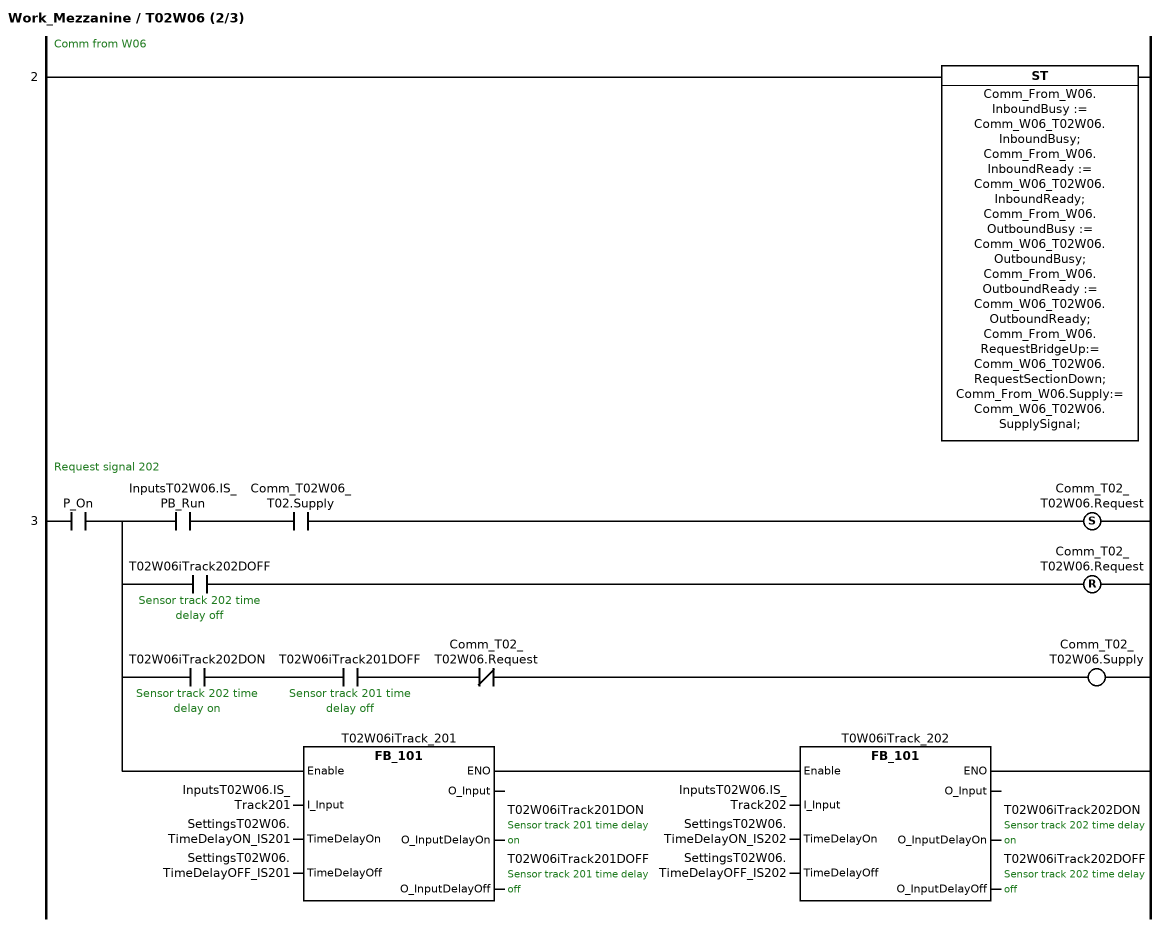
(* [picture p102: Work_Mezzanine / T02W06, rungs 2-3] *)
(* Rung 2: Comm from W06 *)
Comm_From_W06.InboundBusy := Comm_W06_T02W06.InboundBusy;
Comm_From_W06.InboundReady := Comm_W06_T02W06.InboundReady;
Comm_From_W06.OutboundBusy := Comm_W06_T02W06.OutboundBusy;
Comm_From_W06.OutboundReady := Comm_W06_T02W06.OutboundReady;
Comm_From_W06.RequestBridgeUp:= Comm_W06_T02W06.RequestSectionDown;
Comm_From_W06.Supply:= Comm_W06_T02W06.SupplySignal;
(* Rung 3: Request signal 202 *)
IF P_On AND InputsT02W06.IS_PB_Run AND Comm_T02W06_T02.Supply THEN
    Comm_T02_T02W06.Request := TRUE;
END_IF;
IF P_On AND T02W06iTrack202DOFF THEN Comm_T02_T02W06.Request := FALSE; END_IF;
Comm_T02_T02W06.Supply := P_On AND T02W06iTrack202DON AND T02W06iTrack201DOFF AND NOT Comm_T02_T02W06.Request;
T02W06iTrack_201(Enable := P_On, I_Input := InputsT02W06.IS_Track201, TimeDelayOn := SettingsT02W06.TimeDelayON_IS201, TimeDelayOff := SettingsT02W06.TimeDelayOFF_IS201, O_InputDelayOn => T02W06iTrack201DON, O_InputDelayOff => T02W06iTrack201DOFF);
T0W06iTrack_202(Enable := T02W06iTrack_201.ENO, I_Input := InputsT02W06.IS_Track202, TimeDelayOn := SettingsT02W06.TimeDelayON_IS202, TimeDelayOff := SettingsT02W06.TimeDelayOFF_IS202, O_InputDelayOn => T02W06iTrack202DON, O_InputDelayOff => T02W06iTrack202DOFF);

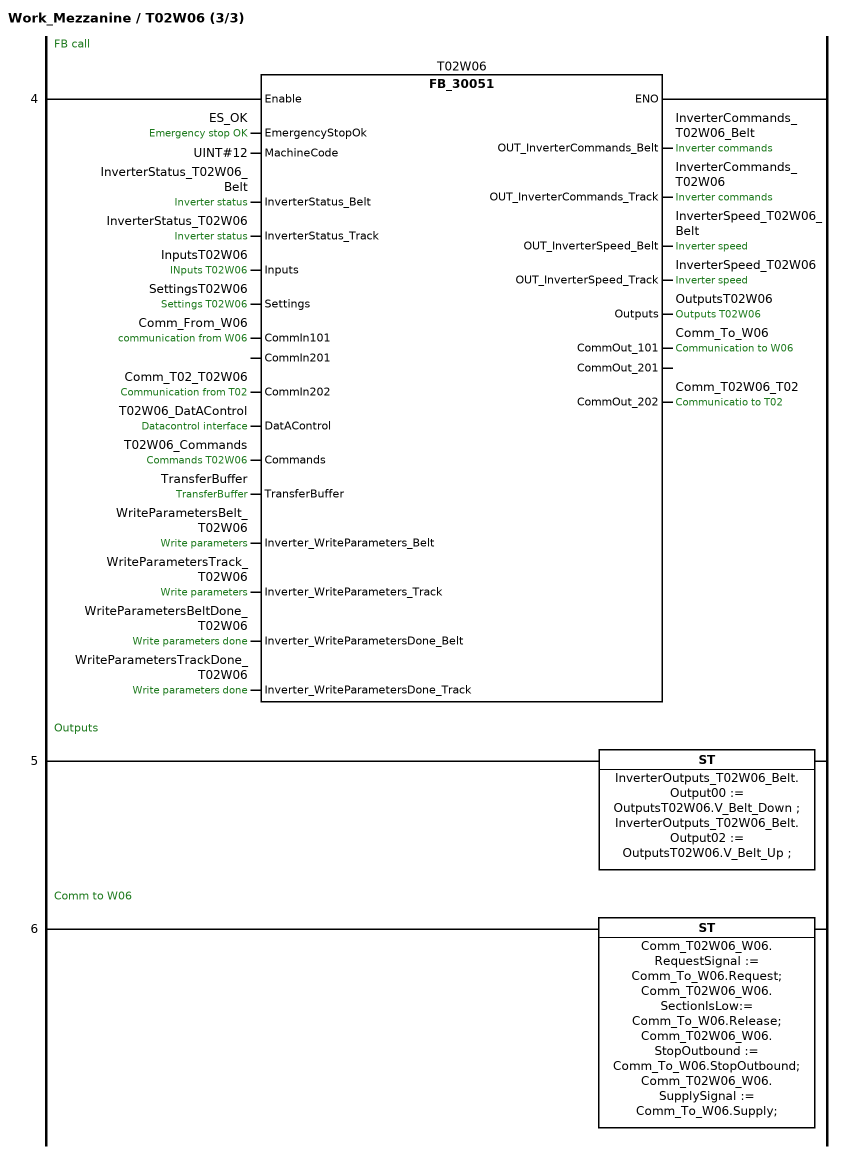
(* Rung 4: FB call *)
T02W06(Enable := TRUE, EmergencyStopOk := ES_OK, MachineCode := UINT#12, InverterStatus_Belt := InverterStatus_T02W06_Belt, InverterStatus_Track := InverterStatus_T02W06, Inputs := InputsT02W06, Settings := SettingsT02W06, CommIn101 := Comm_From_W06, CommIn202 := Comm_T02_T02W06, DatAControl := T02W06_DatAControl, Commands := T02W06_Commands, TransferBuffer := TransferBuffer, Inverter_WriteParameters_Belt := WriteParametersBelt_T02W06, Inverter_WriteParameters_Track := WriteParametersTrack_T02W06, Inverter_WriteParametersDone_Belt := WriteParametersBeltDone_T02W06, Inverter_WriteParametersDone_Track := WriteParametersTrackDone_T02W06, OUT_InverterCommands_Belt => InverterCommands_T02W06_Belt, OUT_InverterCommands_Track => InverterCommands_T02W06, OUT_InverterSpeed_Belt => InverterSpeed_T02W06_Belt, OUT_InverterSpeed_Track => InverterSpeed_T02W06, Outputs => OutputsT02W06, CommOut_101 => Comm_To_W06, CommOut_202 => Comm_T02W06_T02);
(* Rung 5: Outputs *)
InverterOutputs_T02W06_Belt.Output00 := OutputsT02W06.V_Belt_Down ;
InverterOutputs_T02W06_Belt.Output02 := OutputsT02W06.V_Belt_Up ;
(* Rung 6: Comm to W06 *)
Comm_T02W06_W06.RequestSignal := Comm_To_W06.Request;
Comm_T02W06_W06.SectionIsLow:= Comm_To_W06.Release;
Comm_T02W06_W06.StopOutbound := Comm_To_W06.StopOutbound;
Comm_T02W06_W06.SupplySignal := Comm_To_W06.Supply;

(* Section T02W07: ladder, written here as Structured Text *)

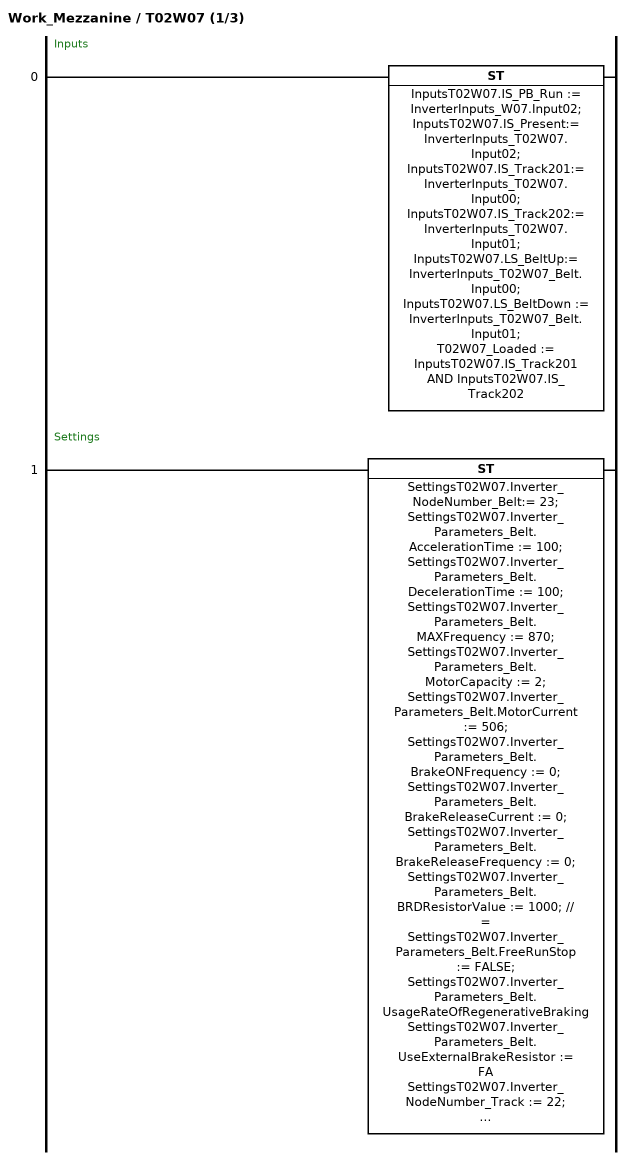
(* Rung 0: Inputs *)
InputsT02W07.IS_PB_Run := InverterInputs_W07.Input02;
InputsT02W07.IS_Present:= InverterInputs_T02W07.Input02;
InputsT02W07.IS_Track201:= InverterInputs_T02W07.Input00;
InputsT02W07.IS_Track202:= InverterInputs_T02W07.Input01;
InputsT02W07.LS_BeltUp:= InverterInputs_T02W07_Belt.Input00;
InputsT02W07.LS_BeltDown := InverterInputs_T02W07_Belt.Input01;

T02W07_Loaded := InputsT02W07.IS_Track201 AND InputsT02W07.IS_Track202;
(* Rung 1: Settings *)
SettingsT02W07.Inverter_NodeNumber_Belt:= 23;
SettingsT02W07.Inverter_Parameters_Belt.AccelerationTime := 100;
SettingsT02W07.Inverter_Parameters_Belt.DecelerationTime := 100;
SettingsT02W07.Inverter_Parameters_Belt.MAXFrequency := 870;
SettingsT02W07.Inverter_Parameters_Belt.MotorCapacity := 2;
SettingsT02W07.Inverter_Parameters_Belt.MotorCurrent := 506;
SettingsT02W07.Inverter_Parameters_Belt.BrakeONFrequency := 0;
SettingsT02W07.Inverter_Parameters_Belt.BrakeReleaseCurrent := 0;
SettingsT02W07.Inverter_Parameters_Belt.BrakeReleaseFrequency := 0;
SettingsT02W07.Inverter_Parameters_Belt.BRDResistorValue := 1000; // = 100,0 ohm, this is the minimum value
SettingsT02W07.Inverter_Parameters_Belt.FreeRunStop := FALSE;
SettingsT02W07.Inverter_Parameters_Belt.UsageRateOfRegenerativeBraking := 0;
SettingsT02W07.Inverter_Parameters_Belt.UseExternalBrakeResistor := FALSE;

SettingsT02W07.Inverter_NodeNumber_Track := 22;
SettingsT02W07.Inverter_Parameters_Track.AccelerationTime := 100;
SettingsT02W07.Inverter_Parameters_Track.DecelerationTime := 100;
SettingsT02W07.Inverter_Parameters_Track.MAXFrequency := 870;
SettingsT02W07.Inverter_Parameters_Track.MotorCapacity := 2;
SettingsT02W07.Inverter_Parameters_Track.MotorCurrent := 506;
SettingsT02W07.Inverter_Parameters_Track.BrakeONFrequency := 0;
SettingsT02W07.Inverter_Parameters_Track.BrakeReleaseCurrent := 0;
SettingsT02W07.Inverter_Parameters_Track.BrakeReleaseFrequency := 0;
SettingsT02W07.Inverter_Parameters_Track.BRDResistorValue := 1000; // = 100,0 ohm, this is the minimum value
SettingsT02W07.Inverter_Parameters_Track.FreeRunStop := FALSE;
SettingsT02W07.Inverter_Parameters_Track.UsageRateOfRegenerativeBraking := 0;
SettingsT02W07.Inverter_Parameters_Track.UseExternalBrakeResistor := FALSE;

SettingsT02W07.ForwardIsInput := TRUE;
SettingsT02W07.MaxSpeed := 3500;
SettingsT02W07.MinSpeed := 1500;
SettingsT02W07.TimeHighSpeed := 100;
SettingsT02W07.MAX_Run_Time := 600;
SettingsT02W07.TimeDelayON_IS201 := 1;
SettingsT02W07.TimeDelayOFF_IS201 := 20;
SettingsT02W07.TimeDelayON_IS202 := 1;
SettingsT02W07.TimeDelayOFF_IS202 := 20;
SettingsT02W07.TimeDelayON_ISPresent := 5;
SettingsT02W07.TimeDelayOFF_ISPresent := 20;
SettingsT02W07.TimeDelayON_LSTrackDown := 20;
SettingsT02W07.TimeDelayON_LSTrackUp := 20;
SettingsT02W07.TrackDirection := T02W07_Direction;
SettingsT02W07.UsePushButton := FALSE;
SettingsT02W07.UseInstructionTrack := TRUE;
SettingsT02W07.MaxSpeedBelt := 5000;
SettingsT02W07.MinSpeedBelt :=3500;
SettingsT02W07.TimeHighSpeedBelt := 120;
SettingsT02W07.HardwareCodeBuffer:= 201;
SettingsT02W07.DoTransferInbound_101:= TRUE;
SettingsT02W07.DoTransferOutbound_101:= TRUE;
SettingsT02W07.DoTransferInbound201_Buffer:= FALSE; // Must be false as soon as BoweryOS and Dat-A-Control 
SettingsT02W07.DoTransferOutbound201_Buffer:= TRUE;
SettingsT02W07.DoTransferInbound202_Buffer:= TRUE;
SettingsT02W07.DoTransferOutbound202_Buffer := FALSE;
SettingsT02W07.DoubleSolenoidValve:= TRUE;

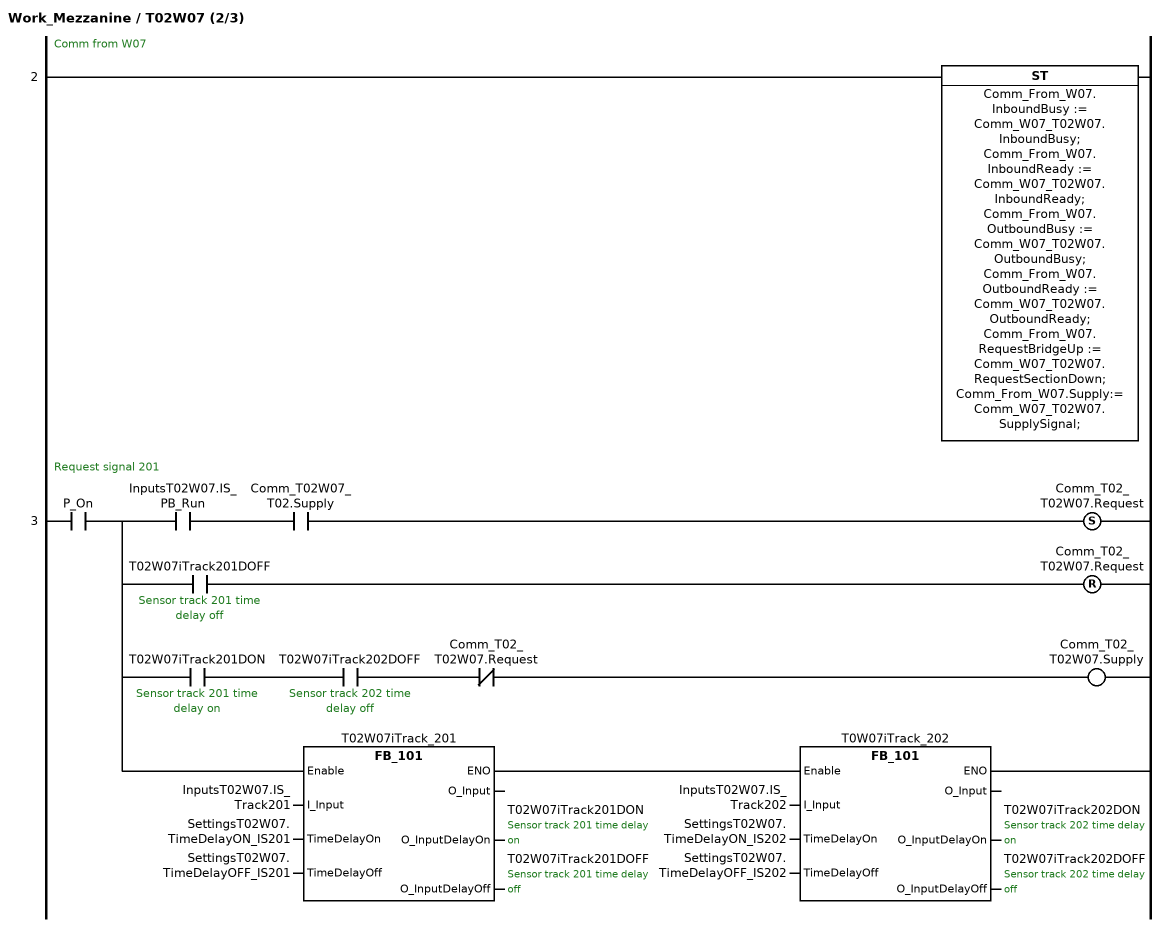
(* Rung 2: Comm from W07 *)
Comm_From_W07.InboundBusy := Comm_W07_T02W07.InboundBusy;
Comm_From_W07.InboundReady := Comm_W07_T02W07.InboundReady;
Comm_From_W07.OutboundBusy := Comm_W07_T02W07.OutboundBusy;
Comm_From_W07.OutboundReady := Comm_W07_T02W07.OutboundReady;
Comm_From_W07.RequestBridgeUp := Comm_W07_T02W07.RequestSectionDown;
Comm_From_W07.Supply:= Comm_W07_T02W07.SupplySignal;
(* Rung 3: Request signal 201 *)
IF P_On AND InputsT02W07.IS_PB_Run AND Comm_T02W07_T02.Supply THEN
    Comm_T02_T02W07.Request := TRUE;
END_IF;
IF P_On AND T02W07iTrack201DOFF THEN Comm_T02_T02W07.Request := FALSE; END_IF;
Comm_T02_T02W07.Supply := P_On AND T02W07iTrack201DON AND T02W07iTrack202DOFF AND NOT Comm_T02_T02W07.Request;
T02W07iTrack_201(Enable := P_On, I_Input := InputsT02W07.IS_Track201, TimeDelayOn := SettingsT02W07.TimeDelayON_IS201, TimeDelayOff := SettingsT02W07.TimeDelayOFF_IS201, O_InputDelayOn => T02W07iTrack201DON, O_InputDelayOff => T02W07iTrack201DOFF);
T0W07iTrack_202(Enable := T02W07iTrack_201.ENO, I_Input := InputsT02W07.IS_Track202, TimeDelayOn := SettingsT02W07.TimeDelayON_IS202, TimeDelayOff := SettingsT02W07.TimeDelayOFF_IS202, O_InputDelayOn => T02W07iTrack202DON, O_InputDelayOff => T02W07iTrack202DOFF);

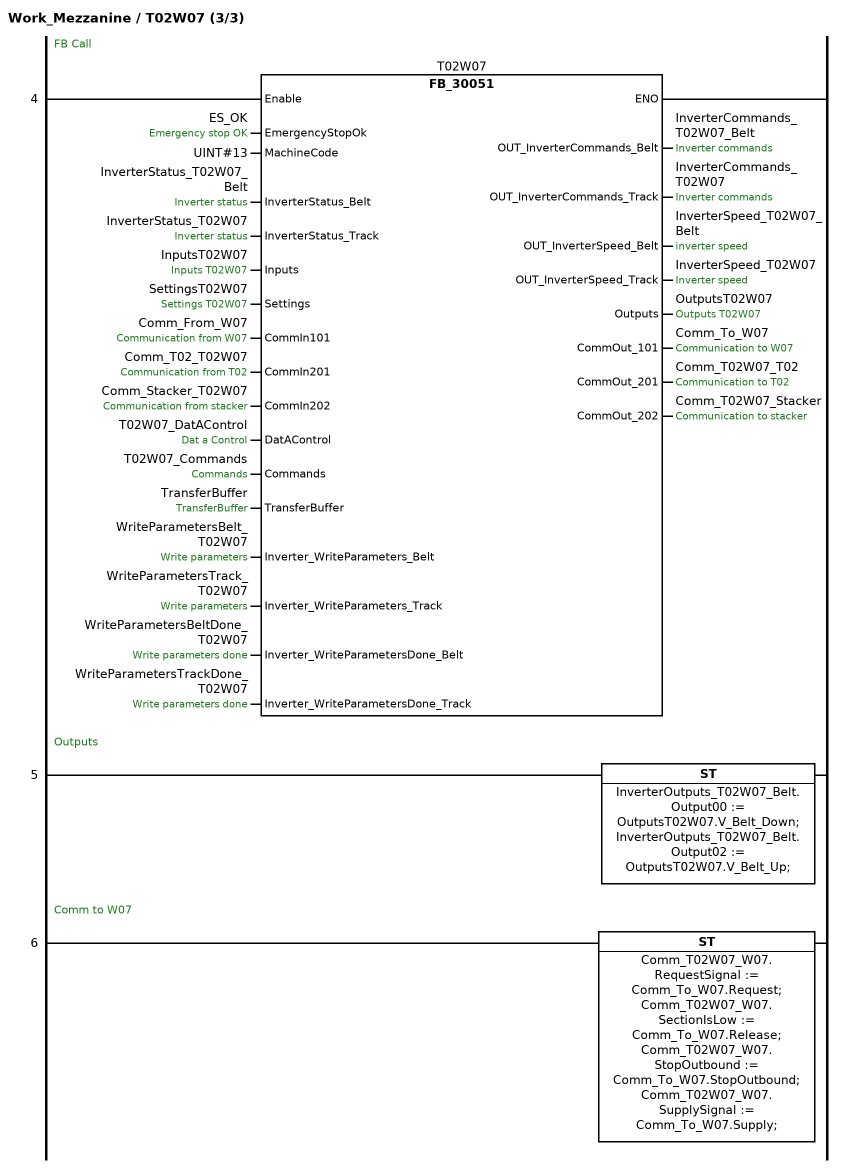
(* Rung 4: FB Call *)
T02W07(Enable := TRUE, EmergencyStopOk := ES_OK, MachineCode := UINT#13, InverterStatus_Belt := InverterStatus_T02W07_Belt, InverterStatus_Track := InverterStatus_T02W07, Inputs := InputsT02W07, Settings := SettingsT02W07, CommIn101 := Comm_From_W07, CommIn201 := Comm_T02_T02W07, CommIn202 := Comm_Stacker_T02W07, DatAControl := T02W07_DatAControl, Commands := T02W07_Commands, TransferBuffer := TransferBuffer, Inverter_WriteParameters_Belt := WriteParametersBelt_T02W07, Inverter_WriteParameters_Track := WriteParametersTrack_T02W07, Inverter_WriteParametersDone_Belt := WriteParametersBeltDone_T02W07, Inverter_WriteParametersDone_Track := WriteParametersTrackDone_T02W07, OUT_InverterCommands_Belt => InverterCommands_T02W07_Belt, OUT_InverterCommands_Track => InverterCommands_T02W07, OUT_InverterSpeed_Belt => InverterSpeed_T02W07_Belt, OUT_InverterSpeed_Track => InverterSpeed_T02W07, Outputs => OutputsT02W07, CommOut_101 => Comm_To_W07, CommOut_201 => Comm_T02W07_T02, CommOut_202 => Comm_T02W07_Stacker);
(* Rung 5: Outputs *)
InverterOutputs_T02W07_Belt.Output00 := OutputsT02W07.V_Belt_Down;
InverterOutputs_T02W07_Belt.Output02 := OutputsT02W07.V_Belt_Up;
(* Rung 6: Comm to W07 *)
Comm_T02W07_W07.RequestSignal := Comm_To_W07.Request;
Comm_T02W07_W07.SectionIsLow := Comm_To_W07.Release;
Comm_T02W07_W07.StopOutbound := Comm_To_W07.StopOutbound;
Comm_T02W07_W07.SupplySignal := Comm_To_W07.Supply;

(* Section W06: ladder, written here as Structured Text *)

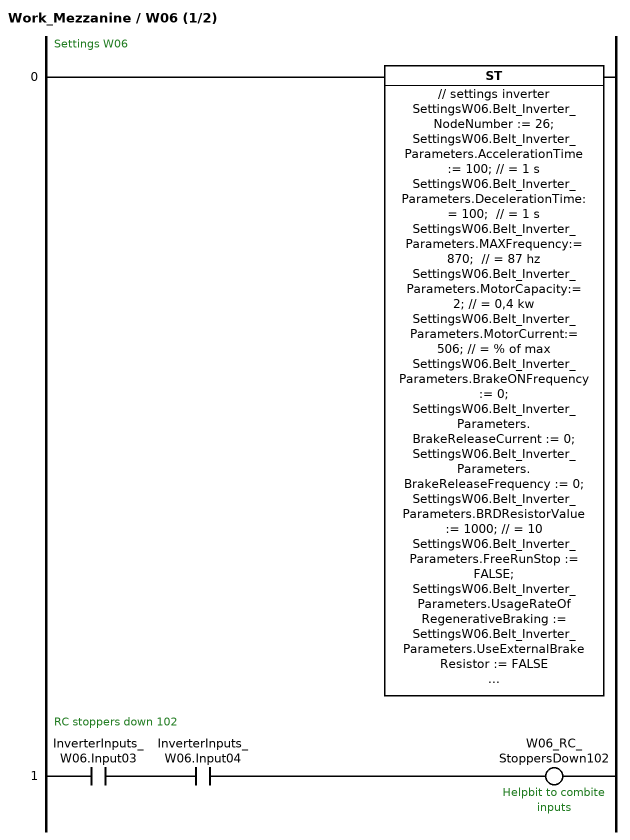
(* Rung 0: Settings W06 *)
// settings inverter
SettingsW06.Belt_Inverter_NodeNumber := 26;
SettingsW06.Belt_Inverter_Parameters.AccelerationTime := 100; // = 1 second
SettingsW06.Belt_Inverter_Parameters.DecelerationTime:= 100;  // = 1 second
SettingsW06.Belt_Inverter_Parameters.MAXFrequency:= 870;  // = 87 hz
SettingsW06.Belt_Inverter_Parameters.MotorCapacity:= 2; // = 0,4 kw
SettingsW06.Belt_Inverter_Parameters.MotorCurrent:= 506; // = % of maximum current
SettingsW06.Belt_Inverter_Parameters.BrakeONFrequency := 0;
SettingsW06.Belt_Inverter_Parameters.BrakeReleaseCurrent := 0;
SettingsW06.Belt_Inverter_Parameters.BrakeReleaseFrequency := 0;
SettingsW06.Belt_Inverter_Parameters.BRDResistorValue := 1000; // = 100,0 ohm, this is the minimum value
SettingsW06.Belt_Inverter_Parameters.FreeRunStop := FALSE;
SettingsW06.Belt_Inverter_Parameters.UsageRateOfRegenerativeBraking := 0;
SettingsW06.Belt_Inverter_Parameters.UseExternalBrakeResistor := FALSE;

SettingsW06.Belt_Max_Run_Time:= 1800;
SettingsW06.Belt_Speed_Max := 5300;
SettingsW06.Belt_Speed_Min := 3500;
SettingsW06.Belt_Speed_Outbound101:= 5000;
SettingsW06.Belt_Speed_Outbound102 := 4600;
SettingsW06.TimeDelayOFF_RS101:= 10;
SettingsW06.TimeDelayON_RS101:= 10;
SettingsW06.TimeDelayOFF_RS102:= 2;
SettingsW06.TimeDelayON_RS102:= 2;
SettingsW06.Time_Belt_Fast := 170;
SettingsW06.DoNotCheckSensors:=TRUE;
SettingsW06.NoInstructionInbound101:= FALSE;
SettingsW06.NoInstructionInbound102:= TRUE;
SettingsW06.Stopper_102:= TRUE;
(* Rung 1: RC stoppers down 102 *)
W06_RC_StoppersDown102 := InverterInputs_W06.Input03 AND InverterInputs_W06.Input04;

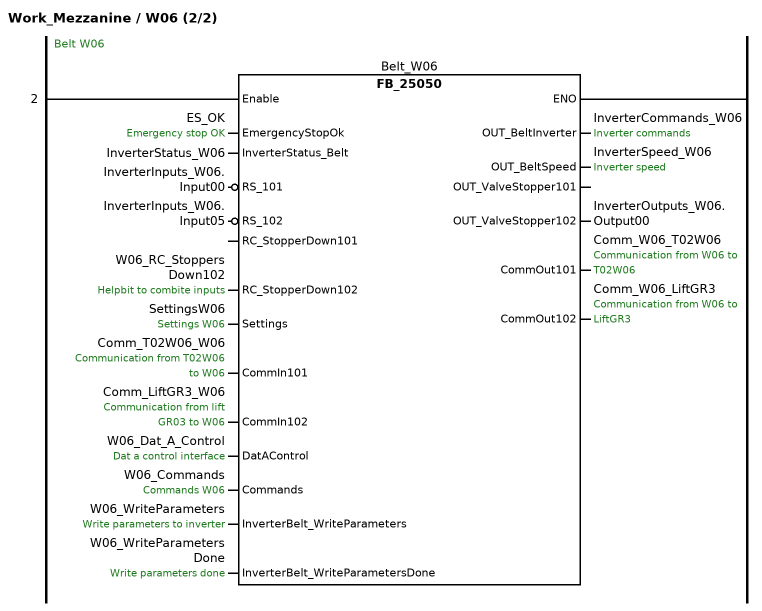
(* Rung 2: Belt W06 *)
Belt_W06(Enable := TRUE, EmergencyStopOk := ES_OK, InverterStatus_Belt := InverterStatus_W06, RS_101 := NOT InverterInputs_W06.Input00, RS_102 := NOT InverterInputs_W06.Input05, RC_StopperDown102 := W06_RC_StoppersDown102, Settings := SettingsW06, CommIn101 := Comm_T02W06_W06, CommIn102 := Comm_LiftGR3_W06, DatAControl := W06_Dat_A_Control, Commands := W06_Commands, InverterBelt_WriteParameters := W06_WriteParameters, InverterBelt_WriteParametersDone := W06_WriteParametersDone, OUT_BeltInverter => InverterCommands_W06, OUT_BeltSpeed => InverterSpeed_W06, OUT_ValveStopper102 => InverterOutputs_W06.Output00, CommOut101 => Comm_W06_T02W06, CommOut102 => Comm_W06_LiftGR3);

(* Section W07: ladder, written here as Structured Text *)

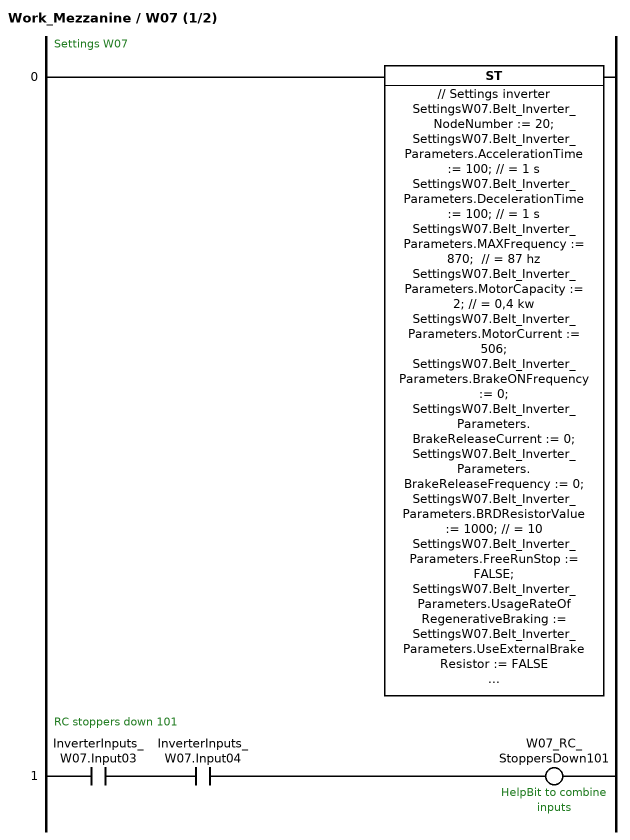
(* Rung 0: Settings W07 *)
// Settings inverter
SettingsW07.Belt_Inverter_NodeNumber := 20;
SettingsW07.Belt_Inverter_Parameters.AccelerationTime := 100; // = 1 second
SettingsW07.Belt_Inverter_Parameters.DecelerationTime := 100; // = 1 second
SettingsW07.Belt_Inverter_Parameters.MAXFrequency := 870;  // = 87 hz
SettingsW07.Belt_Inverter_Parameters.MotorCapacity := 2; // = 0,4 kw
SettingsW07.Belt_Inverter_Parameters.MotorCurrent := 506;
SettingsW07.Belt_Inverter_Parameters.BrakeONFrequency := 0;
SettingsW07.Belt_Inverter_Parameters.BrakeReleaseCurrent := 0;
SettingsW07.Belt_Inverter_Parameters.BrakeReleaseFrequency := 0;
SettingsW07.Belt_Inverter_Parameters.BRDResistorValue := 1000; // = 100,0 ohm, this is the minimum value
SettingsW07.Belt_Inverter_Parameters.FreeRunStop := FALSE;
SettingsW07.Belt_Inverter_Parameters.UsageRateOfRegenerativeBraking := 0;
SettingsW07.Belt_Inverter_Parameters.UseExternalBrakeResistor := FALSE;

SettingsW07.Belt_Max_Run_Time := 1800;
SettingsW07.Belt_Speed_Max := 5300;
SettingsW07.Belt_Speed_Min :=3500;
SettingsW07.Belt_Speed_Outbound101 := 4600;
SettingsW07.Belt_Speed_Outbound102 := 5000;
SettingsW07.TimeDelayOFF_RS101 := 2;
SettingsW07.TimeDelayON_RS101 := 2;
SettingsW07.TimeDelayOFF_RS102 := 10;
SettingsW07.TimeDelayON_RS102 := 10;
SettingsW07.Time_Belt_Fast := 170;
SettingsW07.DoNotCheckSensors := TRUE;
SettingsW07.NoInstructionInbound101 := TRUE;
SettingsW07.NoInstructionInbound102 := FALSE;
SettingsW07.Stopper_101:= TRUE;
(* Rung 1: RC stoppers down 101 *)
W07_RC_StoppersDown101 := InverterInputs_W07.Input03 AND InverterInputs_W07.Input04;

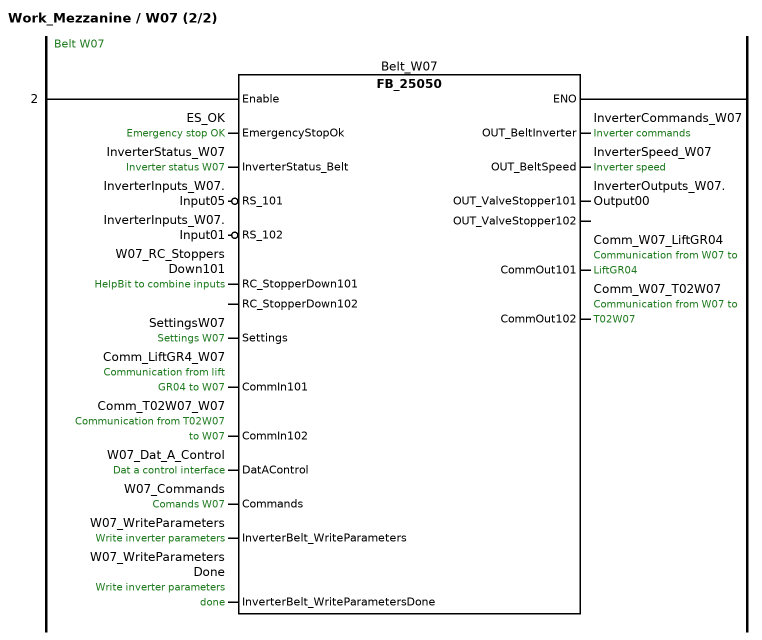
(* Rung 2: Belt W07 *)
Belt_W07(Enable := TRUE, EmergencyStopOk := ES_OK, InverterStatus_Belt := InverterStatus_W07, RS_101 := NOT InverterInputs_W07.Input05, RS_102 := NOT InverterInputs_W07.Input01, RC_StopperDown101 := W07_RC_StoppersDown101, Settings := SettingsW07, CommIn101 := Comm_LiftGR4_W07, CommIn102 := Comm_T02W07_W07, DatAControl := W07_Dat_A_Control, Commands := W07_Commands, InverterBelt_WriteParameters := W07_WriteParameters, InverterBelt_WriteParametersDone := W07_WriteParametersDone, OUT_BeltInverter => InverterCommands_W07, OUT_BeltSpeed => InverterSpeed_W07, OUT_ValveStopper101 => InverterOutputs_W07.Output00, CommOut101 => Comm_W07_LiftGR04, CommOut102 => Comm_W07_T02W07);

(* Section Stacker: ladder, written here as Structured Text *)

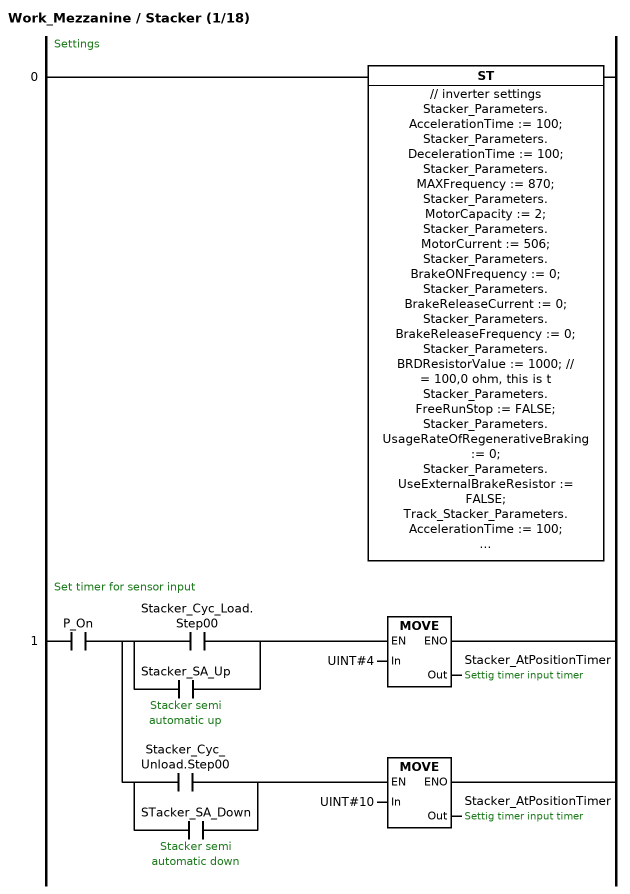
(* Rung 0: Settings *)
// inverter settings
Stacker_Parameters.AccelerationTime := 100;
Stacker_Parameters.DecelerationTime := 100;
Stacker_Parameters.MAXFrequency := 870;
Stacker_Parameters.MotorCapacity := 2;
Stacker_Parameters.MotorCurrent := 506;
Stacker_Parameters.BrakeONFrequency := 0;
Stacker_Parameters.BrakeReleaseCurrent := 0;
Stacker_Parameters.BrakeReleaseFrequency := 0;
Stacker_Parameters.BRDResistorValue := 1000; // = 100,0 ohm, this is the minimum value
Stacker_Parameters.FreeRunStop := FALSE;
Stacker_Parameters.UsageRateOfRegenerativeBraking := 0;
Stacker_Parameters.UseExternalBrakeResistor := FALSE;

Track_Stacker_Parameters.AccelerationTime := 100;
Track_Stacker_Parameters.DecelerationTime := 100;
Track_Stacker_Parameters.MAXFrequency := 870;
Track_Stacker_Parameters.MotorCapacity := 2;
Track_Stacker_Parameters.MotorCurrent := 506;
Track_Stacker_Parameters.BrakeONFrequency := 0;
Track_Stacker_Parameters.BrakeReleaseCurrent := 0;
Track_Stacker_Parameters.BrakeReleaseFrequency := 0;
Track_Stacker_Parameters.BRDResistorValue := 1000; // = 100,0 ohm, this is the minimum value
Track_Stacker_Parameters.FreeRunStop := FALSE;
Track_Stacker_Parameters.UsageRateOfRegenerativeBraking := 0;
Track_Stacker_Parameters.UseExternalBrakeResistor := FALSE;

// Stacker
Stacker_BrakeReleaseFreq := 750; // 1000 = 10Hz
Stacker_BoostTime := 44; // Delay time maxpeed before goto lower speeds
(* Rung 1: Set timer for sensor input *)
IF P_On AND (Stacker_Cyc_Load.Step00 OR Stacker_SA_Up) THEN Stacker_AtPositionTimer := UINT#4; END_IF;
IF P_On AND (Stacker_Cyc_Unload.Step00 OR STacker_SA_Down) THEN
    Stacker_AtPositionTimer := UINT#10;
END_IF;

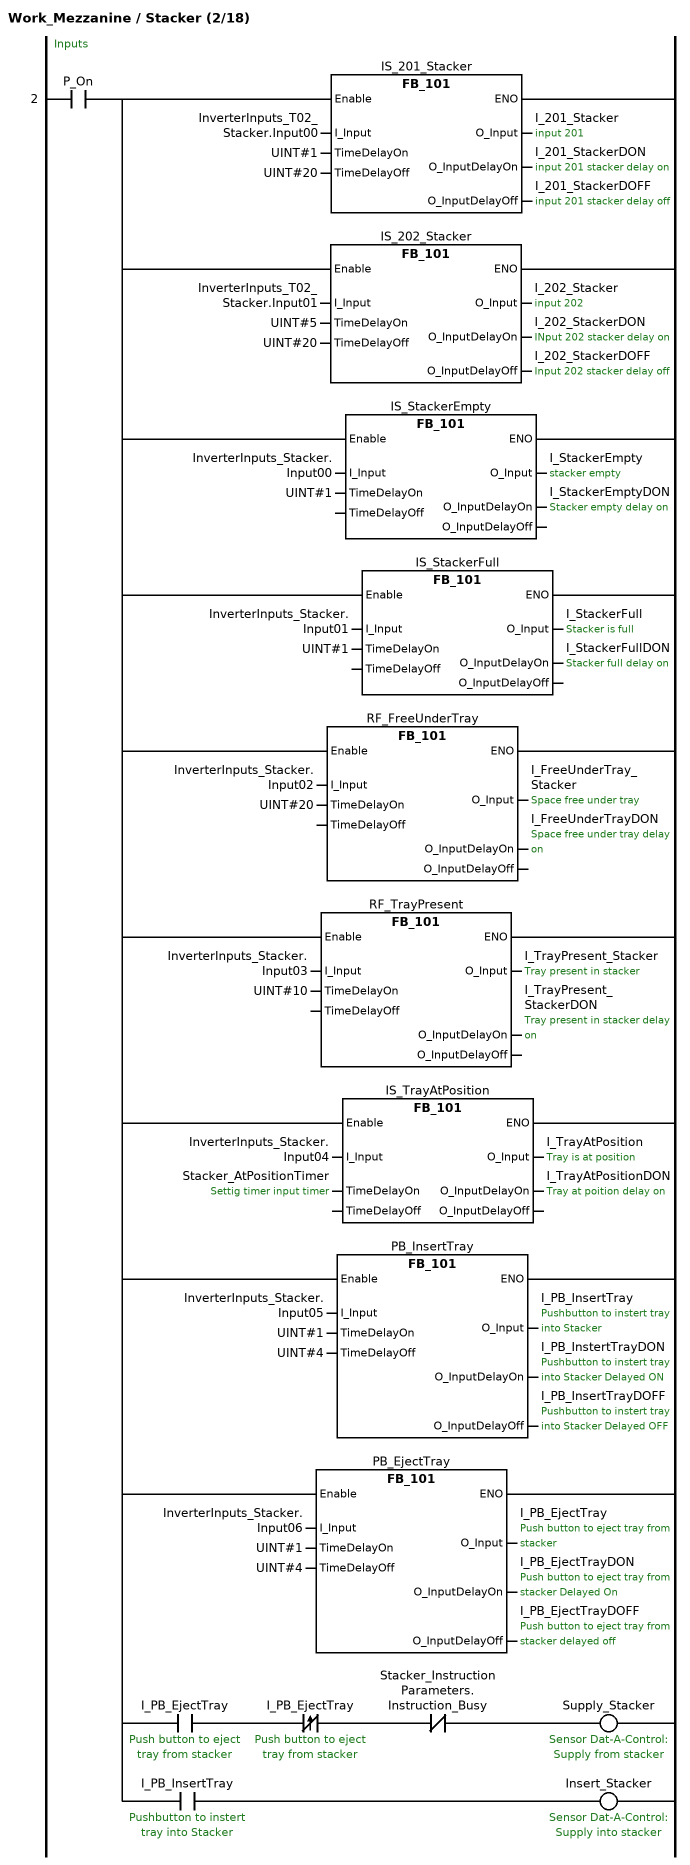
(* Rung 2: Inputs *)
IS_201_Stacker(Enable := P_On, I_Input := InverterInputs_T02_Stacker.Input00, TimeDelayOn := UINT#1, TimeDelayOff := UINT#20, O_Input => I_201_Stacker, O_InputDelayOn => I_201_StackerDON, O_InputDelayOff => I_201_StackerDOFF);
IS_202_Stacker(Enable := P_On, I_Input := InverterInputs_T02_Stacker.Input01, TimeDelayOn := UINT#5, TimeDelayOff := UINT#20, O_Input => I_202_Stacker, O_InputDelayOn => I_202_StackerDON, O_InputDelayOff => I_202_StackerDOFF);
IS_StackerEmpty(Enable := P_On, I_Input := InverterInputs_Stacker.Input00, TimeDelayOn := UINT#1, O_Input => I_StackerEmpty, O_InputDelayOn => I_StackerEmptyDON);
IS_StackerFull(Enable := P_On, I_Input := InverterInputs_Stacker.Input01, TimeDelayOn := UINT#1, O_Input => I_StackerFull, O_InputDelayOn => I_StackerFullDON);
RF_FreeUnderTray(Enable := P_On, I_Input := InverterInputs_Stacker.Input02, TimeDelayOn := UINT#20, O_Input => I_FreeUnderTray_Stacker, O_InputDelayOn => I_FreeUnderTrayDON);
RF_TrayPresent(Enable := P_On, I_Input := InverterInputs_Stacker.Input03, TimeDelayOn := UINT#10, O_Input => I_TrayPresent_Stacker, O_InputDelayOn => I_TrayPresent_StackerDON);
IS_TrayAtPosition(Enable := P_On, I_Input := InverterInputs_Stacker.Input04, TimeDelayOn := Stacker_AtPositionTimer, O_Input => I_TrayAtPosition, O_InputDelayOn => I_TrayAtPositionDON);
PB_InsertTray(Enable := P_On, I_Input := InverterInputs_Stacker.Input05, TimeDelayOn := UINT#1, TimeDelayOff := UINT#4, O_Input => I_PB_InsertTray, O_InputDelayOn => I_PB_InstertTrayDON, O_InputDelayOff => I_PB_InsertTrayDOFF);
PB_EjectTray(Enable := P_On, I_Input := InverterInputs_Stacker.Input06, TimeDelayOn := UINT#1, TimeDelayOff := UINT#4, O_Input => I_PB_EjectTray, O_InputDelayOn => I_PB_EjectTrayDON, O_InputDelayOff => I_PB_EjectTrayDOFF);
_e1(CLK := I_PB_EjectTray);
Supply_Stacker := P_On AND I_PB_EjectTray AND NOT _e1.Q AND NOT Stacker_InstructionParameters.Instruction_Busy;
Insert_Stacker := P_On AND I_PB_InsertTray;

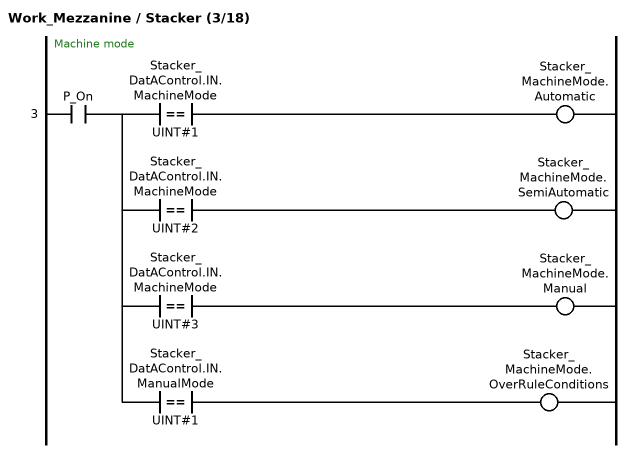
(* Rung 3: Machine mode *)
Stacker_MachineMode.Automatic := P_On AND (Stacker_DatAControl.IN.MachineMode = UINT#1);
Stacker_MachineMode.SemiAutomatic := P_On AND (Stacker_DatAControl.IN.MachineMode = UINT#2);
Stacker_MachineMode.Manual := P_On AND (Stacker_DatAControl.IN.MachineMode = UINT#3);
Stacker_MachineMode.OverRuleConditions := P_On AND (Stacker_DatAControl.IN.ManualMode = UINT#1);

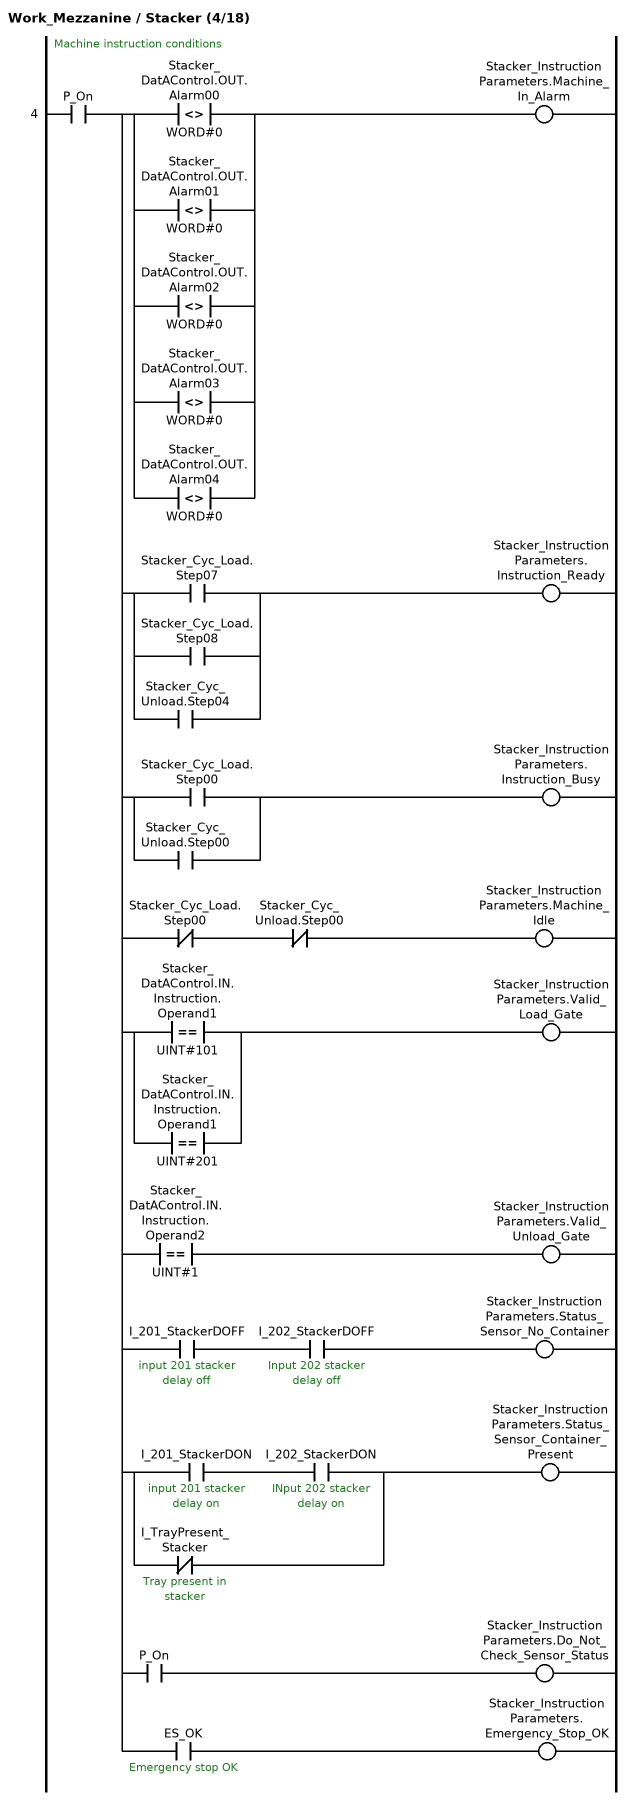
(* Rung 4: Machine instruction conditions *)
Stacker_InstructionParameters.Machine_In_Alarm := P_On AND ((Stacker_DatAControl.OUT.Alarm00 <> WORD#0) OR (Stacker_DatAControl.OUT.Alarm01 <> WORD#0) OR (Stacker_DatAControl.OUT.Alarm02 <> WORD#0) OR (Stacker_DatAControl.OUT.Alarm03 <> WORD#0) OR (Stacker_DatAControl.OUT.Alarm04 <> WORD#0));
Stacker_InstructionParameters.Instruction_Ready := P_On AND (Stacker_Cyc_Load.Step07 OR Stacker_Cyc_Load.Step08 OR Stacker_Cyc_Unload.Step04);
Stacker_InstructionParameters.Instruction_Busy := P_On AND (Stacker_Cyc_Load.Step00 OR Stacker_Cyc_Unload.Step00);
Stacker_InstructionParameters.Machine_Idle := P_On AND NOT Stacker_Cyc_Load.Step00 AND NOT Stacker_Cyc_Unload.Step00;
Stacker_InstructionParameters.Valid_Load_Gate := P_On AND ((Stacker_DatAControl.IN.Instruction.Operand1 = UINT#101) OR (Stacker_DatAControl.IN.Instruction.Operand1 = UINT#201));
Stacker_InstructionParameters.Valid_Unload_Gate := P_On AND (Stacker_DatAControl.IN.Instruction.Operand2 = UINT#1);
Stacker_InstructionParameters.Status_Sensor_No_Container := P_On AND I_201_StackerDOFF AND I_202_StackerDOFF;
Stacker_InstructionParameters.Status_Sensor_Container_Present := P_On AND ((I_201_StackerDON AND I_202_StackerDON) OR NOT I_TrayPresent_Stacker);
Stacker_InstructionParameters.Do_Not_Check_Sensor_Status := P_On AND P_On;
Stacker_InstructionParameters.Emergency_Stop_OK := P_On AND ES_OK;

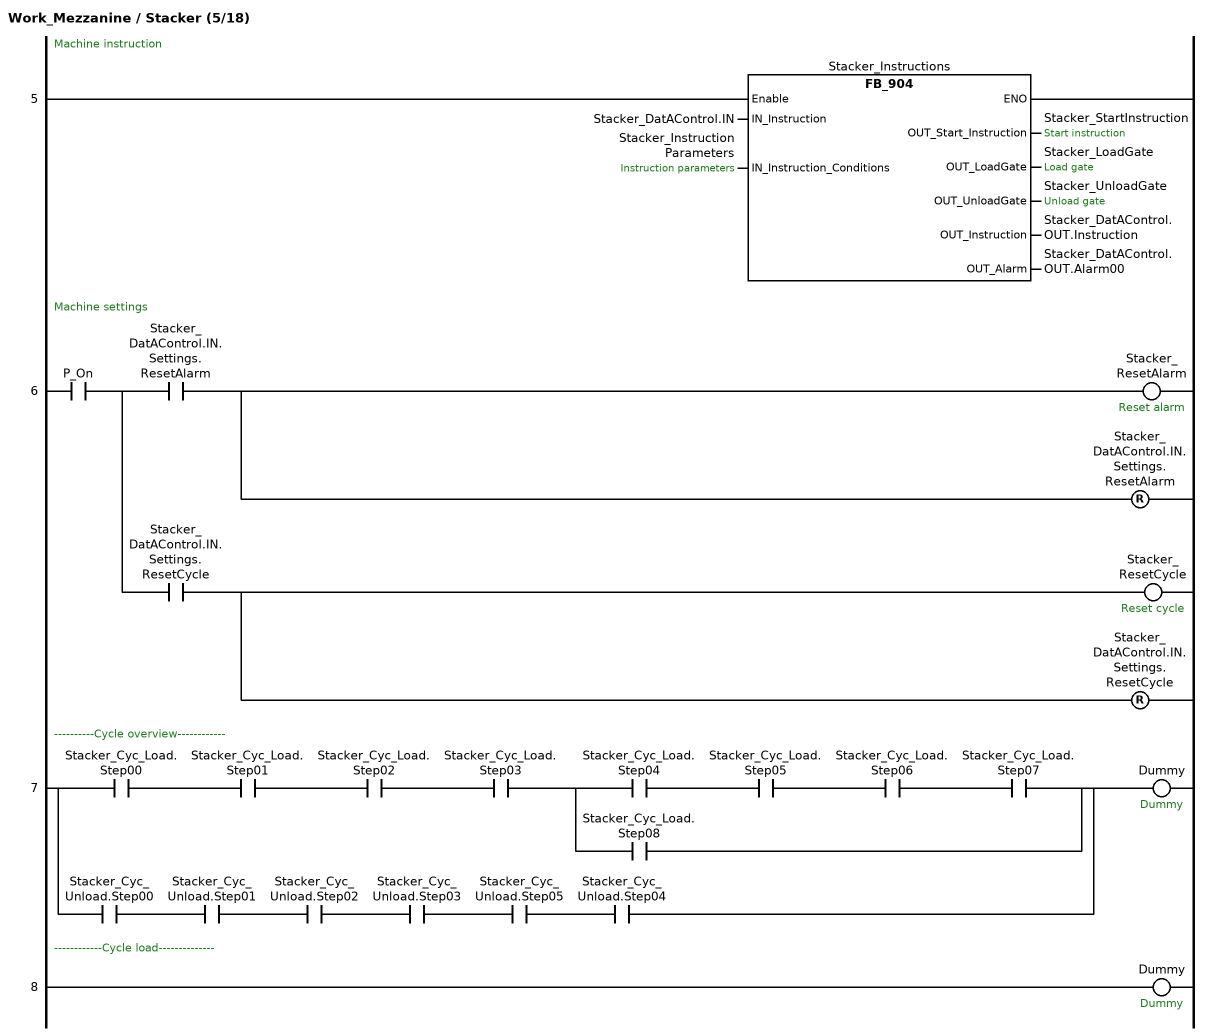
(* Rung 5: Machine instruction *)
Stacker_Instructions(Enable := TRUE, IN_Instruction := Stacker_DatAControl.IN, IN_Instruction_Conditions := Stacker_InstructionParameters, OUT_Start_Instruction => Stacker_StartInstruction, OUT_LoadGate => Stacker_LoadGate, OUT_UnloadGate => Stacker_UnloadGate, OUT_Instruction => Stacker_DatAControl.OUT.Instruction, OUT_Alarm => Stacker_DatAControl.OUT.Alarm00);
(* Rung 6: Machine settings *)
_p2 := P_On AND Stacker_DatAControl.IN.Settings.ResetAlarm;
Stacker_ResetAlarm := _p2;
IF _p2 THEN Stacker_DatAControl.IN.Settings.ResetAlarm := FALSE; END_IF;
_p3 := P_On AND Stacker_DatAControl.IN.Settings.ResetCycle;
Stacker_ResetCycle := _p3;
IF _p3 THEN Stacker_DatAControl.IN.Settings.ResetCycle := FALSE; END_IF;
(* Rung 7: ----------Cycle overview------------ *)
Dummy := (Stacker_Cyc_Load.Step00 AND Stacker_Cyc_Load.Step01 AND Stacker_Cyc_Load.Step02 AND Stacker_Cyc_Load.Step03 AND ((Stacker_Cyc_Load.Step04 AND Stacker_Cyc_Load.Step05 AND Stacker_Cyc_Load.Step06 AND Stacker_Cyc_Load.Step07) OR Stacker_Cyc_Load.Step08)) OR (Stacker_Cyc_Unload.Step00 AND Stacker_Cyc_Unload.Step01 AND Stacker_Cyc_Unload.Step02 AND Stacker_Cyc_Unload.Step03 AND Stacker_Cyc_Unload.Step05 AND Stacker_Cyc_Unload.Step04);
(* Rung 8: ------------Cycle load-------------- *)
Dummy := TRUE;

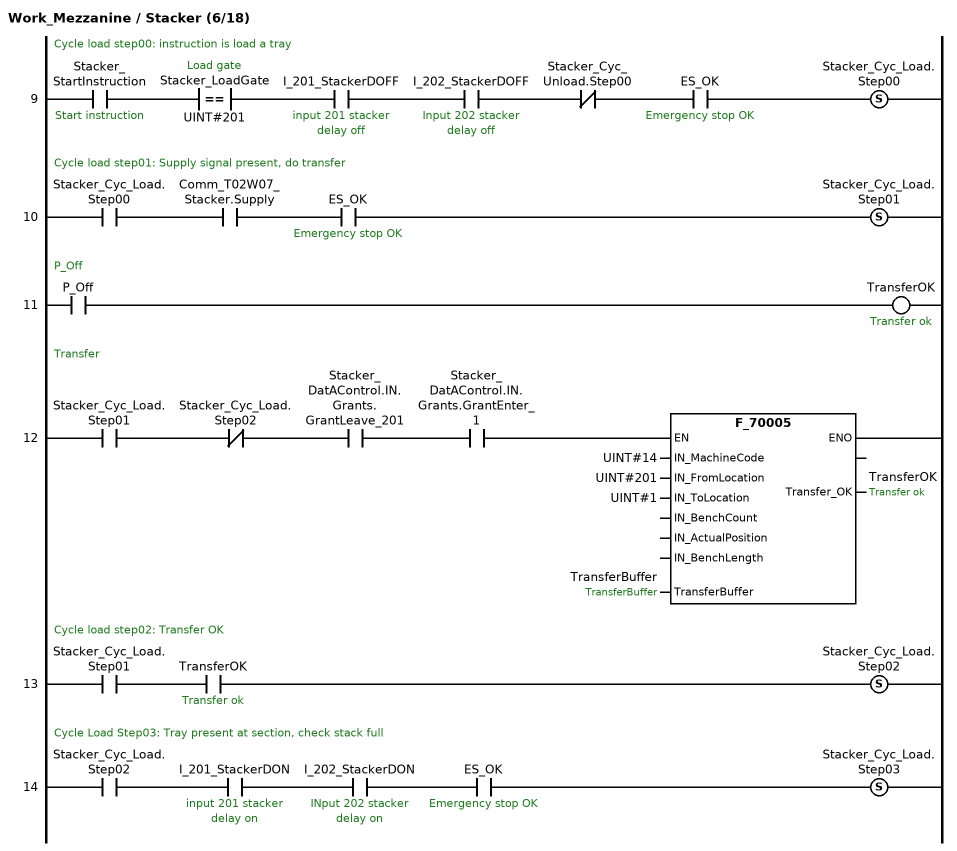
(* Rung 9: Cycle load step00: instruction is load a tray *)
IF Stacker_StartInstruction AND (Stacker_LoadGate = UINT#201) AND I_201_StackerDOFF AND I_202_StackerDOFF AND NOT Stacker_Cyc_Unload.Step00 AND ES_OK THEN
    Stacker_Cyc_Load.Step00 := TRUE;
END_IF;
(* Rung 10: Cycle load step01: Supply signal present, do transfer *)
IF Stacker_Cyc_Load.Step00 AND Comm_T02W07_Stacker.Supply AND ES_OK THEN
    Stacker_Cyc_Load.Step01 := TRUE;
END_IF;
(* Rung 11: P_Off *)
TransferOK := P_Off;
(* Rung 12: Transfer *)
IF Stacker_Cyc_Load.Step01 AND NOT Stacker_Cyc_Load.Step02 AND Stacker_DatAControl.IN.Grants.GrantLeave_201 AND Stacker_DatAControl.IN.Grants.GrantEnter_1 THEN
    F_70005(IN_MachineCode := UINT#14, IN_FromLocation := UINT#201, IN_ToLocation := UINT#1, TransferBuffer := TransferBuffer, Transfer_OK => TransferOK);
END_IF;
(* Rung 13: Cycle load step02: Transfer OK *)
IF Stacker_Cyc_Load.Step01 AND TransferOK THEN Stacker_Cyc_Load.Step02 := TRUE; END_IF;
(* Rung 14: Cycle Load Step03: Tray present at section, check stack full *)
IF Stacker_Cyc_Load.Step02 AND I_201_StackerDON AND I_202_StackerDON AND ES_OK THEN
    Stacker_Cyc_Load.Step03 := TRUE;
END_IF;

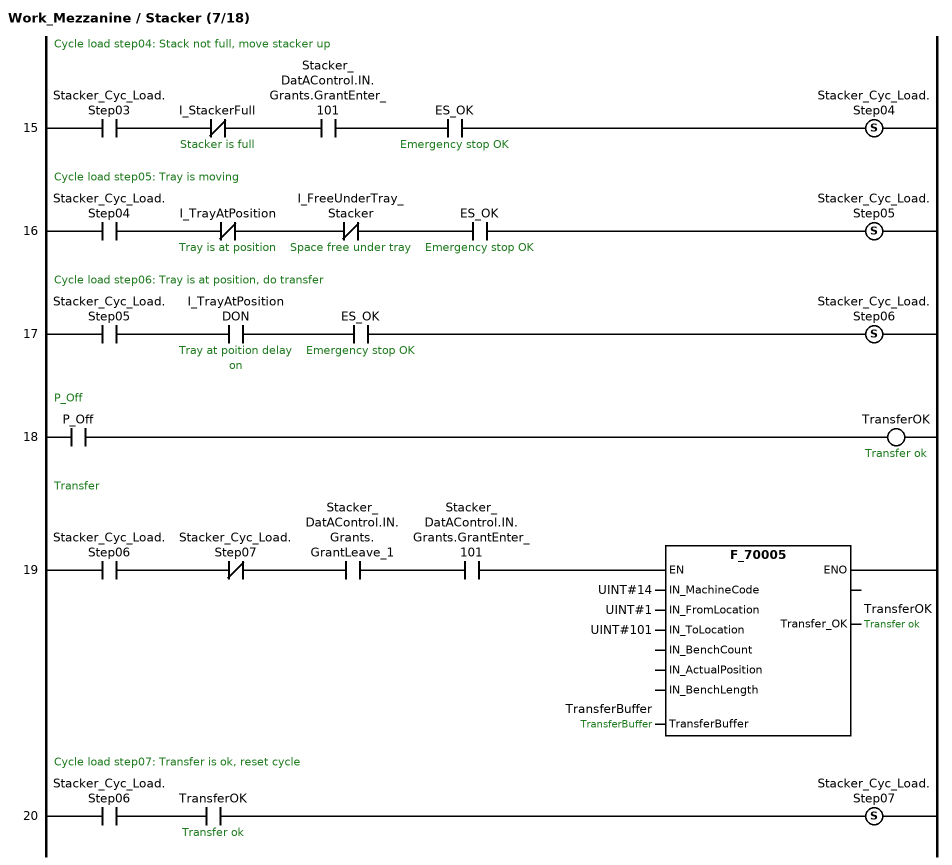
(* Rung 15: Cycle load step04: Stack not full, move stacker up *)
IF Stacker_Cyc_Load.Step03 AND NOT I_StackerFull AND Stacker_DatAControl.IN.Grants.GrantEnter_101 AND ES_OK THEN
    Stacker_Cyc_Load.Step04 := TRUE;
END_IF;
(* Rung 16: Cycle load step05: Tray is moving *)
IF Stacker_Cyc_Load.Step04 AND NOT I_TrayAtPosition AND NOT I_FreeUnderTray_Stacker AND ES_OK THEN
    Stacker_Cyc_Load.Step05 := TRUE;
END_IF;
(* Rung 17: Cycle load step06: Tray is at position, do transfer *)
IF Stacker_Cyc_Load.Step05 AND I_TrayAtPositionDON AND ES_OK THEN Stacker_Cyc_Load.Step06 := TRUE; END_IF;
(* Rung 18: P_Off *)
TransferOK := P_Off;
(* Rung 19: Transfer *)
IF Stacker_Cyc_Load.Step06 AND NOT Stacker_Cyc_Load.Step07 AND Stacker_DatAControl.IN.Grants.GrantLeave_1 AND Stacker_DatAControl.IN.Grants.GrantEnter_101 THEN
    F_70005(IN_MachineCode := UINT#14, IN_FromLocation := UINT#1, IN_ToLocation := UINT#101, TransferBuffer := TransferBuffer, Transfer_OK => TransferOK);
END_IF;
(* Rung 20: Cycle load step07: Transfer is ok, reset cycle *)
IF Stacker_Cyc_Load.Step06 AND TransferOK THEN Stacker_Cyc_Load.Step07 := TRUE; END_IF;

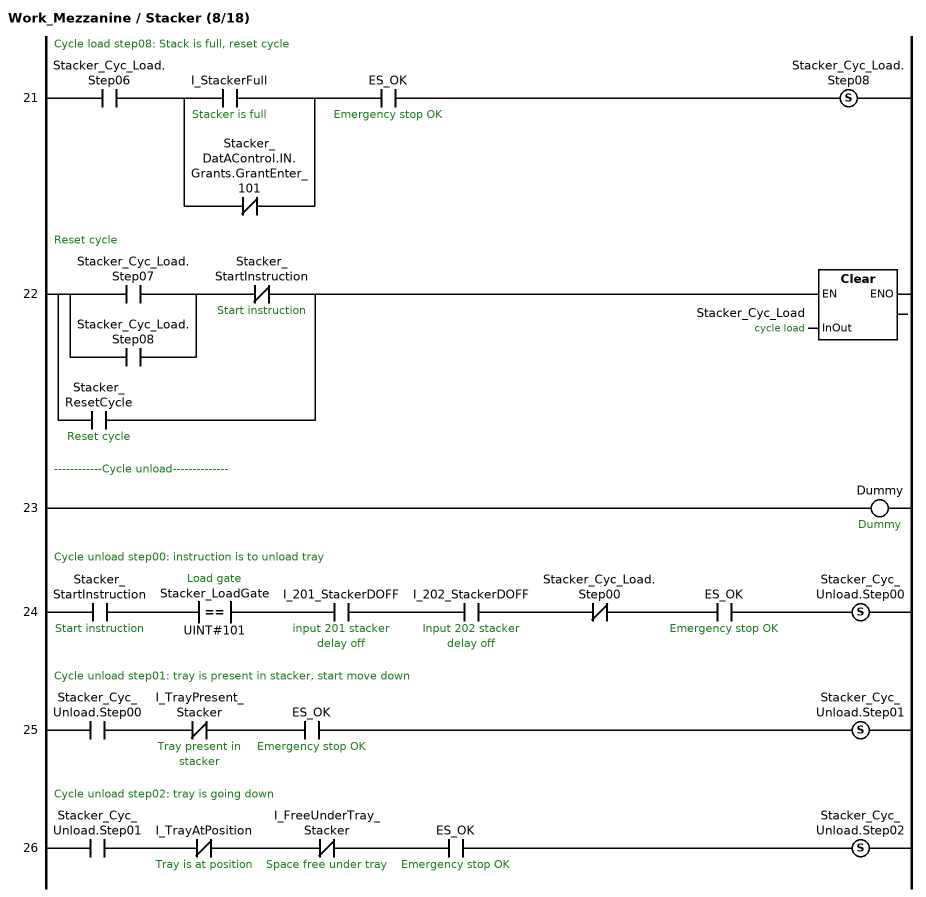
(* Rung 21: Cycle load step08: Stack is full, reset cycle *)
IF Stacker_Cyc_Load.Step06 AND (I_StackerFull OR NOT Stacker_DatAControl.IN.Grants.GrantEnter_101) AND ES_OK THEN
    Stacker_Cyc_Load.Step08 := TRUE;
END_IF;
(* Rung 22: Reset cycle *)
IF ((Stacker_Cyc_Load.Step07 OR Stacker_Cyc_Load.Step08) AND NOT Stacker_StartInstruction) OR Stacker_ResetCycle THEN
    Clear(InOut := Stacker_Cyc_Load);
END_IF;
(* Rung 23: ------------Cycle unload-------------- *)
Dummy := TRUE;
(* Rung 24: Cycle unload step00: instruction is to unload tray *)
IF Stacker_StartInstruction AND (Stacker_LoadGate = UINT#101) AND I_201_StackerDOFF AND I_202_StackerDOFF AND NOT Stacker_Cyc_Load.Step00 AND ES_OK THEN
    Stacker_Cyc_Unload.Step00 := TRUE;
END_IF;
(* Rung 25: Cycle unload step01: tray is present in stacker, start move down *)
IF Stacker_Cyc_Unload.Step00 AND NOT I_TrayPresent_Stacker AND ES_OK THEN
    Stacker_Cyc_Unload.Step01 := TRUE;
END_IF;
(* Rung 26: Cycle unload step02: tray is going down *)
IF Stacker_Cyc_Unload.Step01 AND NOT I_TrayAtPosition AND NOT I_FreeUnderTray_Stacker AND ES_OK THEN
    Stacker_Cyc_Unload.Step02 := TRUE;
END_IF;

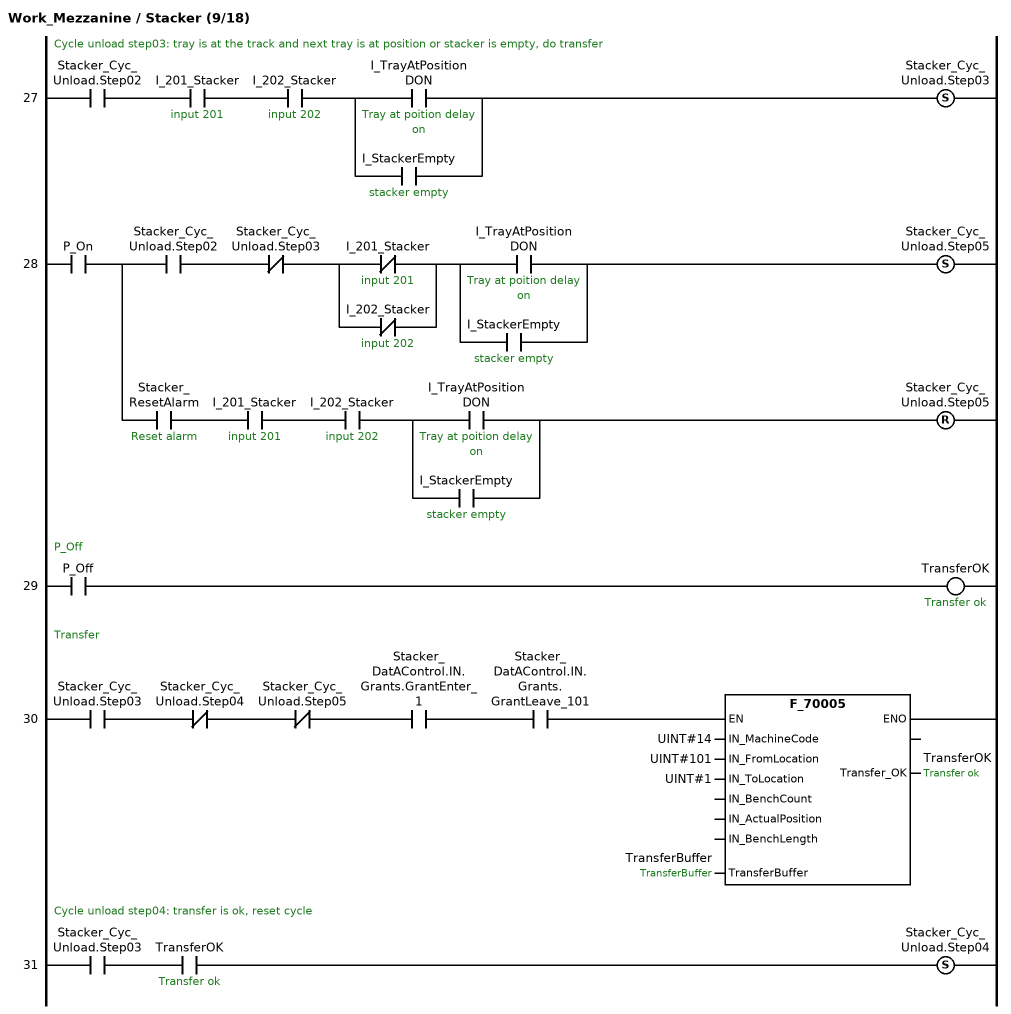
(* Rung 27: Cycle unload step03: tray is at the track and next tray is at position or stacker is empty, do transfer *)
IF Stacker_Cyc_Unload.Step02 AND I_201_Stacker AND I_202_Stacker AND (I_TrayAtPositionDON OR I_StackerEmpty) THEN
    Stacker_Cyc_Unload.Step03 := TRUE;
END_IF;
(* Rung 28 *)
IF P_On AND Stacker_Cyc_Unload.Step02 AND NOT Stacker_Cyc_Unload.Step03 AND (NOT I_201_Stacker OR NOT I_202_Stacker) AND (I_TrayAtPositionDON OR I_StackerEmpty) THEN
    Stacker_Cyc_Unload.Step05 := TRUE;
END_IF;
IF P_On AND Stacker_ResetAlarm AND I_201_Stacker AND I_202_Stacker AND (I_TrayAtPositionDON OR I_StackerEmpty) THEN
    Stacker_Cyc_Unload.Step05 := FALSE;
END_IF;
(* Rung 29: P_Off *)
TransferOK := P_Off;
(* Rung 30: Transfer *)
IF Stacker_Cyc_Unload.Step03 AND NOT Stacker_Cyc_Unload.Step04 AND NOT Stacker_Cyc_Unload.Step05 AND Stacker_DatAControl.IN.Grants.GrantEnter_1 AND Stacker_DatAControl.IN.Grants.GrantLeave_101 THEN
    F_70005(IN_MachineCode := UINT#14, IN_FromLocation := UINT#101, IN_ToLocation := UINT#1, TransferBuffer := TransferBuffer, Transfer_OK => TransferOK);
END_IF;
(* Rung 31: Cycle unload step04: transfer is ok, reset cycle *)
IF Stacker_Cyc_Unload.Step03 AND TransferOK THEN Stacker_Cyc_Unload.Step04 := TRUE; END_IF;

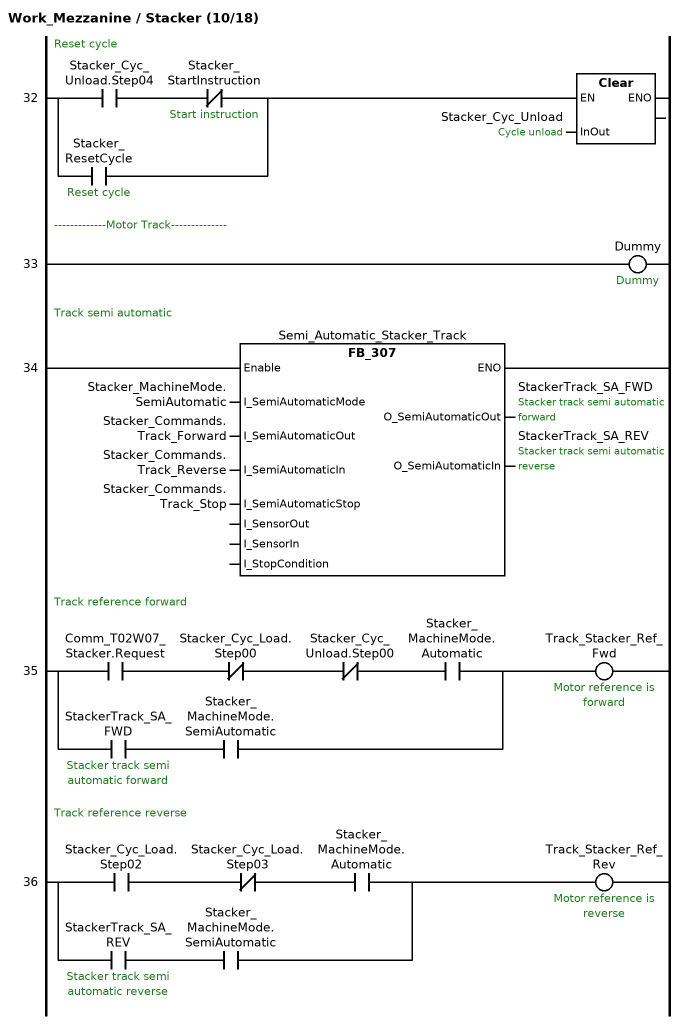
(* Rung 32: Reset cycle *)
IF (Stacker_Cyc_Unload.Step04 AND NOT Stacker_StartInstruction) OR Stacker_ResetCycle THEN
    Clear(InOut := Stacker_Cyc_Unload);
END_IF;
(* Rung 33: -------------Motor Track-------------- *)
Dummy := TRUE;
(* Rung 34: Track semi automatic *)
Semi_Automatic_Stacker_Track(Enable := TRUE, I_SemiAutomaticMode := Stacker_MachineMode.SemiAutomatic, I_SemiAutomaticOut := Stacker_Commands.Track_Forward, I_SemiAutomaticIn := Stacker_Commands.Track_Reverse, I_SemiAutomaticStop := Stacker_Commands.Track_Stop, O_SemiAutomaticOut => StackerTrack_SA_FWD, O_SemiAutomaticIn => StackerTrack_SA_REV);
(* Rung 35: Track reference forward *)
Track_Stacker_Ref_Fwd := (Comm_T02W07_Stacker.Request AND NOT Stacker_Cyc_Load.Step00 AND NOT Stacker_Cyc_Unload.Step00 AND Stacker_MachineMode.Automatic) OR (StackerTrack_SA_FWD AND Stacker_MachineMode.SemiAutomatic);
(* Rung 36: Track reference reverse *)
Track_Stacker_Ref_Rev := (Stacker_Cyc_Load.Step02 AND NOT Stacker_Cyc_Load.Step03 AND Stacker_MachineMode.Automatic) OR (StackerTrack_SA_REV AND Stacker_MachineMode.SemiAutomatic);

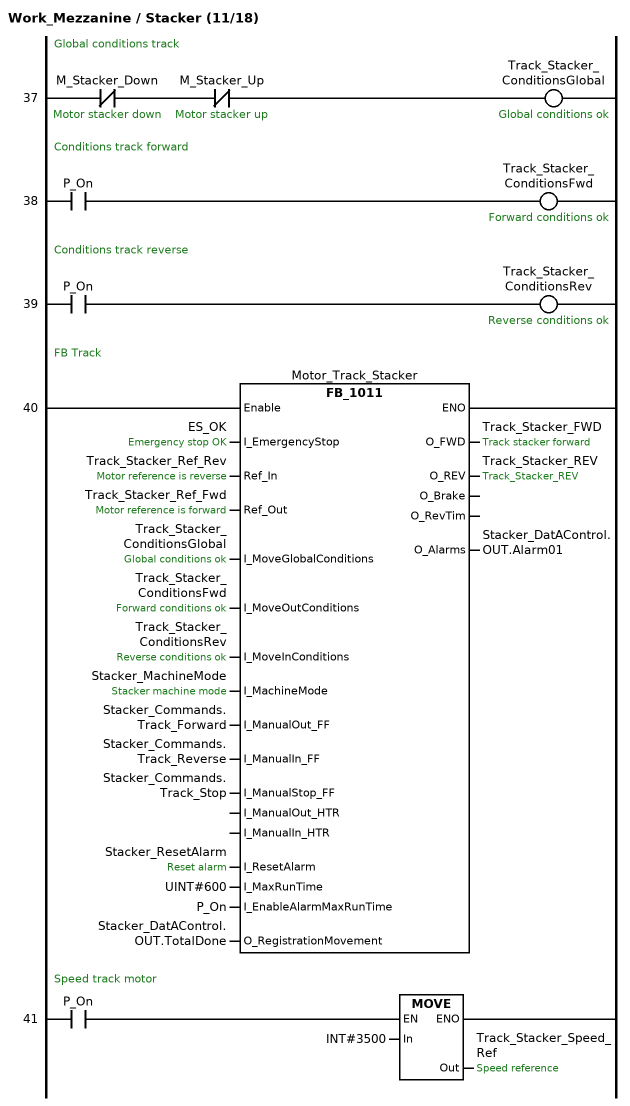
(* Rung 37: Global conditions track *)
Track_Stacker_ConditionsGlobal := NOT M_Stacker_Down AND NOT M_Stacker_Up;
(* Rung 38: Conditions track forward *)
Track_Stacker_ConditionsFwd := P_On;
(* Rung 39: Conditions track reverse *)
Track_Stacker_ConditionsRev := P_On;
(* Rung 40: FB Track *)
Motor_Track_Stacker(Enable := TRUE, I_EmergencyStop := ES_OK, Ref_In := Track_Stacker_Ref_Rev, Ref_Out := Track_Stacker_Ref_Fwd, I_MoveGlobalConditions := Track_Stacker_ConditionsGlobal, I_MoveOutConditions := Track_Stacker_ConditionsFwd, I_MoveInConditions := Track_Stacker_ConditionsRev, I_MachineMode := Stacker_MachineMode, I_ManualOut_FF := Stacker_Commands.Track_Forward, I_ManualIn_FF := Stacker_Commands.Track_Reverse, I_ManualStop_FF := Stacker_Commands.Track_Stop, I_ResetAlarm := Stacker_ResetAlarm, I_MaxRunTime := UINT#600, I_EnableAlarmMaxRunTime := P_On, O_RegistrationMovement := Stacker_DatAControl.OUT.TotalDone, O_FWD => Track_Stacker_FWD, O_REV => Track_Stacker_REV, O_Alarms => Stacker_DatAControl.OUT.Alarm01);
(* Rung 41: Speed track motor *)
IF P_On THEN Track_Stacker_Speed_Ref := INT#3500; END_IF;

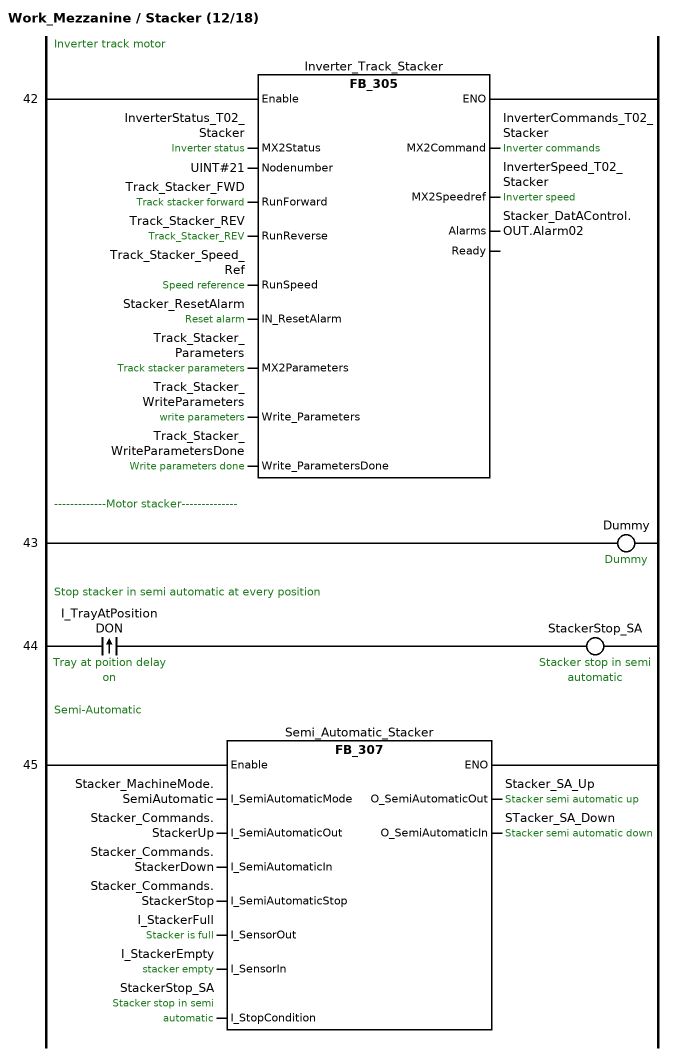
(* Rung 42: Inverter track motor *)
Inverter_Track_Stacker(Enable := TRUE, MX2Status := InverterStatus_T02_Stacker, Nodenumber := UINT#21, RunForward := Track_Stacker_FWD, RunReverse := Track_Stacker_REV, RunSpeed := Track_Stacker_Speed_Ref, IN_ResetAlarm := Stacker_ResetAlarm, MX2Parameters := Track_Stacker_Parameters, Write_Parameters := Track_Stacker_WriteParameters, Write_ParametersDone := Track_Stacker_WriteParametersDone, MX2Command => InverterCommands_T02_Stacker, MX2Speedref => InverterSpeed_T02_Stacker, Alarms => Stacker_DatAControl.OUT.Alarm02);
(* Rung 43: -------------Motor stacker-------------- *)
Dummy := TRUE;
(* Rung 44: Stop stacker in semi automatic at every position *)
_e4(CLK := I_TrayAtPositionDON);
StackerStop_SA := _e4.Q;
(* Rung 45: Semi-Automatic *)
Semi_Automatic_Stacker(Enable := TRUE, I_SemiAutomaticMode := Stacker_MachineMode.SemiAutomatic, I_SemiAutomaticOut := Stacker_Commands.StackerUp, I_SemiAutomaticIn := Stacker_Commands.StackerDown, I_SemiAutomaticStop := Stacker_Commands.StackerStop, I_SensorOut := I_StackerFull, I_SensorIn := I_StackerEmpty, I_StopCondition := StackerStop_SA, O_SemiAutomaticOut => Stacker_SA_Up, O_SemiAutomaticIn => STacker_SA_Down);

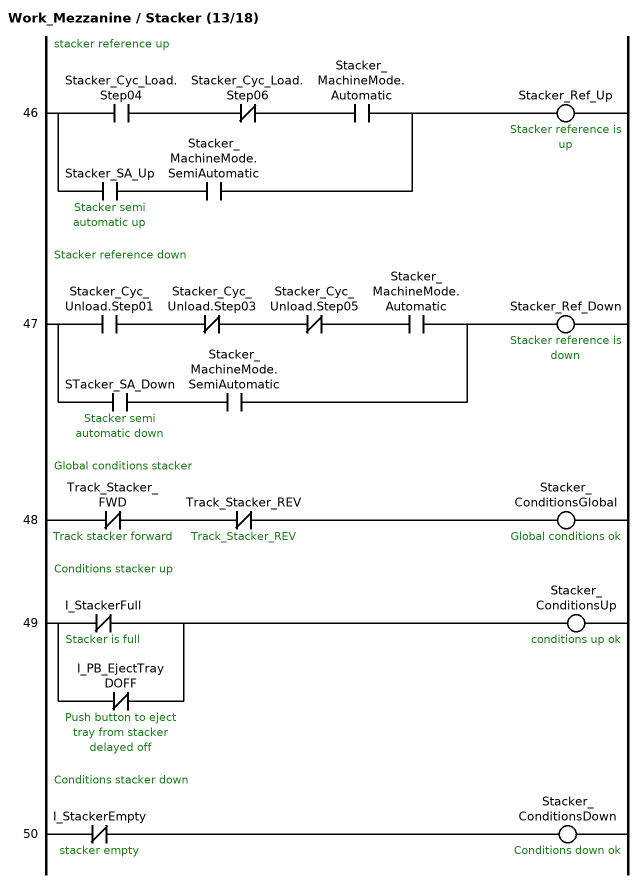
(* Rung 46: stacker reference up *)
Stacker_Ref_Up := (Stacker_Cyc_Load.Step04 AND NOT Stacker_Cyc_Load.Step06 AND Stacker_MachineMode.Automatic) OR (Stacker_SA_Up AND Stacker_MachineMode.SemiAutomatic);
(* Rung 47: Stacker reference down *)
Stacker_Ref_Down := (Stacker_Cyc_Unload.Step01 AND NOT Stacker_Cyc_Unload.Step03 AND NOT Stacker_Cyc_Unload.Step05 AND Stacker_MachineMode.Automatic) OR (STacker_SA_Down AND Stacker_MachineMode.SemiAutomatic);
(* Rung 48: Global conditions stacker *)
Stacker_ConditionsGlobal := NOT Track_Stacker_FWD AND NOT Track_Stacker_REV;
(* Rung 49: Conditions stacker up *)
Stacker_ConditionsUp := NOT I_StackerFull OR NOT I_PB_EjectTrayDOFF;
(* Rung 50: Conditions stacker down *)
Stacker_ConditionsDown := NOT I_StackerEmpty;

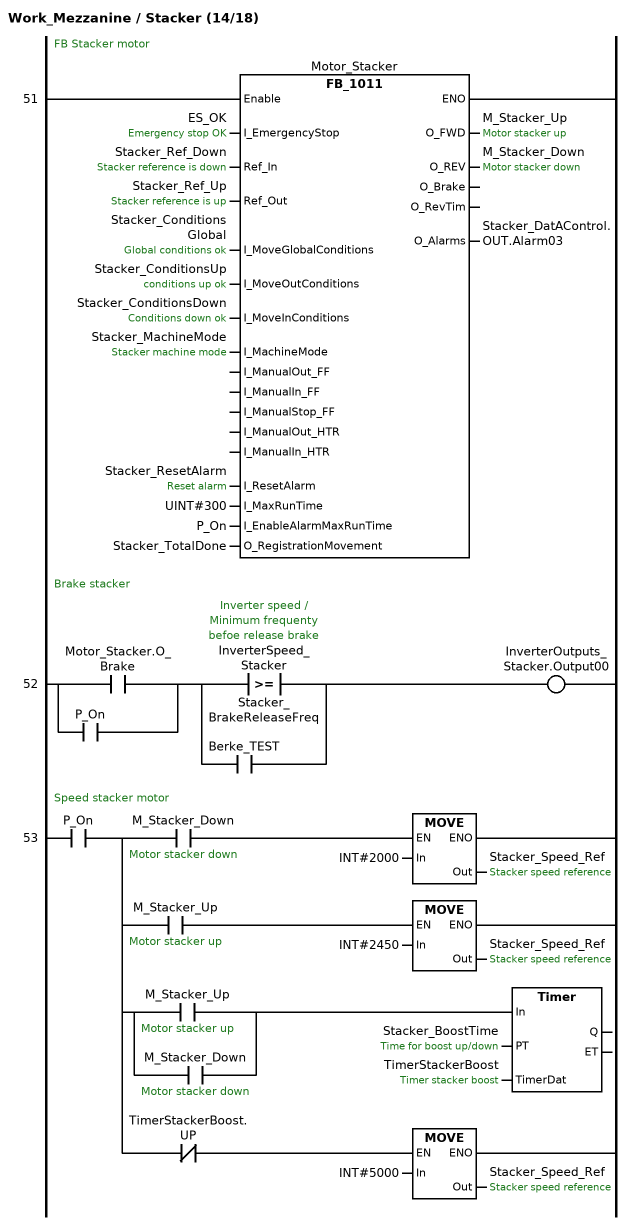
(* Rung 51: FB Stacker motor *)
Motor_Stacker(Enable := TRUE, I_EmergencyStop := ES_OK, Ref_In := Stacker_Ref_Down, Ref_Out := Stacker_Ref_Up, I_MoveGlobalConditions := Stacker_ConditionsGlobal, I_MoveOutConditions := Stacker_ConditionsUp, I_MoveInConditions := Stacker_ConditionsDown, I_MachineMode := Stacker_MachineMode, I_ResetAlarm := Stacker_ResetAlarm, I_MaxRunTime := UINT#300, I_EnableAlarmMaxRunTime := P_On, O_RegistrationMovement := Stacker_TotalDone, O_FWD => M_Stacker_Up, O_REV => M_Stacker_Down, O_Alarms => Stacker_DatAControl.OUT.Alarm03);
(* Rung 52: Brake stacker *)
InverterOutputs_Stacker.Output00 := (Motor_Stacker.O_Brake OR P_On) AND ((InverterSpeed_Stacker >= Stacker_BrakeReleaseFreq) OR Berke_TEST);
(* Rung 53: Speed stacker motor *)
IF P_On AND M_Stacker_Down THEN Stacker_Speed_Ref := INT#2000; END_IF;
IF P_On AND M_Stacker_Up THEN Stacker_Speed_Ref := INT#2450; END_IF;
_t5 := Timer(In := P_On AND (M_Stacker_Up OR M_Stacker_Down), PT := Stacker_BoostTime, TimerDat := TimerStackerBoost);
IF P_On AND NOT TimerStackerBoost.UP THEN Stacker_Speed_Ref := INT#5000; END_IF;

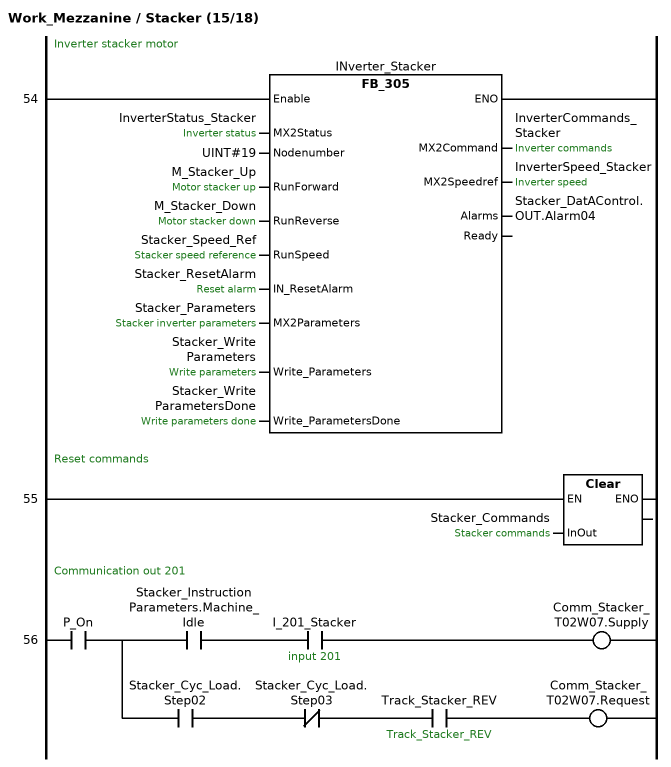
(* Rung 54: Inverter stacker motor *)
INverter_Stacker(Enable := TRUE, MX2Status := InverterStatus_Stacker, Nodenumber := UINT#19, RunForward := M_Stacker_Up, RunReverse := M_Stacker_Down, RunSpeed := Stacker_Speed_Ref, IN_ResetAlarm := Stacker_ResetAlarm, MX2Parameters := Stacker_Parameters, Write_Parameters := Stacker_WriteParameters, Write_ParametersDone := Stacker_WriteParametersDone, MX2Command => InverterCommands_Stacker, MX2Speedref => InverterSpeed_Stacker, Alarms => Stacker_DatAControl.OUT.Alarm04);
(* Rung 55: Reset commands *)
Clear(InOut := Stacker_Commands);
(* Rung 56: Communication out 201 *)
Comm_Stacker_T02W07.Supply := P_On AND Stacker_InstructionParameters.Machine_Idle AND I_201_Stacker;
Comm_Stacker_T02W07.Request := P_On AND Stacker_Cyc_Load.Step02 AND NOT Stacker_Cyc_Load.Step03 AND Track_Stacker_REV;

